FUNCTION_BLOCK FB_Debounce 
VAR_INPUT
	bInput:				BOOL;
	tTime:				TIME;
END_VAR
VAR_OUTPUT
	bValue:				BOOL;
END_VAR
VAR
	fbTimerOn:			Ton;
	fbTimerOff:			Ton;
END_VAR

// https://github.com/PeterZerlauth/Tc3_Component
IF bInput THEN
	fbTimerOn(IN:= TRUE, PT:= tTime);
	fbTimerOff(IN:= FALSE);
	IF fbTimerOn.Q THEN
		bValue:= TRUE;
	END_IF
ELSE
	fbTimerOff(IN:= TRUE, PT:= tTime);
	fbTimerOn(IN:= FALSE);
	IF fbTimerOff.Q THEN
		bValue:= FALSE;
	END_IF	
END_IF

END_FUNCTION_BLOCK

(* stored: Version 1.1.0.1
   POU FB_Debounce: Id {156ff626-5fc6-0a96-33e9-b808df5601eb}, SpecialFunc None *)
